FUNCTION_BLOCK FB_axis
VAR_INPUT
	//bStart							: BOOL;		
END_VAR
VAR_OUTPUT
	power	: ST_McOutputs;	
	resets	: ST_McOutputs;	
	estops	: ST_McOutputs;	
	stops	: ST_McOutputs;	
	driveResets	: ST_McOutputs;	
	diags		: ST_McOutputs;	
	diagNumber	: UDINT;
	moveRels  : ST_McOutputs;
	moveVels  : ST_McOutputs;
	moveAbses : ST_McOutputs;
	readVels	 : ST_McOutputs;
	actVel								: LREAL;
	readPoses	 : ST_McOutputs;
	actPos								: LREAL;
END_VAR
VAR_IN_OUT
	Axis: AXIS_REF;
END_VAR
VAR
	//eState		: axisState;
	mcPower		: MC_Power;
	mcReset		: MC_Reset;
	//mcDriveReset: FB_SoEReset;
	mcMoveAbs	: MC_MoveAbsolute;
	mcStop		: MC_Stop;
	mcMoveRel	: MC_MoveRelative;
	//mcReadDiag	: FB_SoEReadDiagNumber;
	mcReadVel	: MC_ReadActualVelocity;
	mcReadPos	: MC_ReadActualPosition;
	mcMoveVel	: MC_MoveVelocity;
END_VAR

(*Axis.ReadStatus();

IF axis.Status.Error THEN
	eState := ERROR;	
END_IF
	

CASE eState OF
	INIT:
	           //gHW.errAck := TRUE; 
	    mcReset.Execute := FALSE;
		mcPower.Enable := FALSE;
		mcPower.Enable_Negative:= FALSE;
		mcPower.Enable_Positive:= FALSE;
		eState := ENABLE;
		
	ENABLE:		
	         //gHW.errAck := FALSE;
		mcPower.Enable := TRUE;
		mcPower.Enable_Negative:= TRUE;
		mcPower.Enable_Positive:= TRUE;
		IF mcPower.Status THEN
			eState := READY;
		END_IF	
		
	READY:
		IF bStart THEN
			eState:= ESTOP;
		END_IF
		
	ESTOP:		
		mcMoveRel.Distance := 100;
		mcMoveRel.Velocity := 100;
		mcMoveRel.Execute := TRUE;
		IF mcMoveRel.Done THEN
			mcMoveRel.Execute := FALSE;
			eState := READY;
		END_IF	
		
	ERROR:
		mcReset.Execute := TRUE;
		         //gHW.errAck := TRUE; 
		//mcPower.Enable := FALSE;
		//mcPower.Enable_Negative:= FALSE;
		//mcPower.Enable_Positive:= FALSE;
	    IF mcReset.Done THEN
			mcReset.Execute := FALSE;	
			eState := INIT;
		//eState := DISABLED;
		END_IF
END_CASE	

mcPower(Axis:= Axis);
mcMoveRel(Axis:= Axis);
mcReset(Axis:= Axis);*)

METHOD Enable : BOOL
VAR_INPUT
	bEnable : BOOL;
END_VAR
mcPower(
	Axis := Axis,
	Enable := bEnable,
	Enable_Positive := bEnable,
	Enable_Negative := bEnable,
	BufferMode := MC_Aborting,
	Override := 100,
	Status => power.Done,
	Error => power.Error
);
END_METHOD

METHOD eStop : BOOL
VAR_INPUT
	bExecute : BOOL;
END_VAR
VAR
	EStopDeceleration		: LREAL := 5000;
	EStopJerk				: LREAL := 20000;
END_VAR
mcStop(
	Axis := Axis,
	Execute := bExecute,
	Deceleration := EStopDeceleration,
	Jerk := EStopJerk,
	Done => estops.Done
);
END_METHOD

METHOD MoveAbs : BOOL
VAR_INPUT
	bExecute 			: BOOL;
	targetAngle 		: LREAL;
	velocityIncline		: LREAL;
END_VAR
VAR	
	accelerationIncline						: LREAL := 1000;
	decelerationIncline						: LREAL := 1500;
	jerkIncline								: LREAL;
END_VAR
mcMoveAbs(	
	Axis 		:= Axis,
	Execute 	:= bExecute,	
	Position			:= targetAngle,
	Velocity 			:= velocityIncline,//cali
	Acceleration 		:= accelerationIncline,
	Deceleration 		:= decelerationIncline,
	Jerk 				:= jerkIncline,	
	Done 			=> moveAbses.Done,
	Busy 			=> moveAbses.Busy,
	Active 			=> moveAbses.Active,
	CommandAborted 	=> moveAbses.CommandAborted,
	Error 			=> moveAbses.Error,
	ErrorID 		=> moveAbses.ErrorID,	
);
END_METHOD

METHOD MoveRel : BOOL
VAR_INPUT
	bExecute : BOOL;
	relAngle : LREAL;
END_VAR
VAR
	velocityIncline							: LREAL := 100;
	accelerationIncline						: LREAL := 1000;
	decelerationIncline						: LREAL := 1500;
	jerkIncline								: LREAL;
END_VAR
mcMoveRel(
	Axis := Axis,
	Execute := bExecute,
	Distance			:= relAngle,
	Velocity 			:= velocityIncline,//cali
	Acceleration 		:= accelerationIncline,
	Deceleration 		:= decelerationIncline,
	Jerk 				:= jerkIncline,	
	Done 			=> moveRels.Done,
	Busy 			=> moveRels.Busy,
	Active 			=> moveRels.Active,
	CommandAborted 	=> moveRels.CommandAborted,
	Error 			=> moveRels.Error,
	ErrorID 		=> moveRels.ErrorID
);
END_METHOD

METHOD MoveVel : BOOL
VAR_INPUT
	bExecute 		: BOOL;
	velocity		: LREAL;
	acceleration	: LREAL;
	deceleration	: LREAL;
	jerk			: LREAL;
	Direction		: MC_Direction;
END_VAR
VAR
	//BufferMode: MC_Aborting
END_VAR
mcMoveVel(	
	Axis 		:= Axis,
	Execute 	:= bExecute,		
	Velocity 			:= velocity*1,//speedCalibrationFactorL,//cali
	Acceleration 		:= acceleration,
	Deceleration 		:= deceleration,
	Jerk 				:= jerk,	
	BufferMode 			:= MC_Aborting,
	InVelocity 		=> moveVels.Done,
	Busy 			=> moveVels.Busy,
	Active 			=> moveVels.Active,
	CommandAborted 	=> moveVels.CommandAborted,
	Error 			=> moveVels.Error,
	ErrorID 		=> moveVels.ErrorID,	
);
END_METHOD

METHOD ReadPos : BOOL
VAR_INPUT
	bEnable : BOOL;
END_VAR
mcReadPos (
	Axis := Axis,
	Enable := bEnable,
	Busy => readPoses.Busy,
	Position => ActPos
	//Error => diagNumberError,
	//AdsErrId => diagNumberAdsErrorID,
	//SercosErrId => diagNumberSercosErrorID 
);
END_METHOD

METHOD ReadVel : BOOL
VAR_INPUT
	bEnable : BOOL;
END_VAR
mcReadVel (
	Axis := Axis,
	Enable := bEnable,
	Busy => readVels.Busy,
	ActualVelocity => ActVel
	//Error => diagNumberError,
	//AdsErrId => diagNumberAdsErrorID,
	//SercosErrId => diagNumberSercosErrorID 
);
END_METHOD

METHOD Reset : BOOL
VAR_INPUT
	bExecute : BOOL;
END_VAR
mcReset(
	Axis := Axis,
	Execute := bExecute,
	Done => resets.Done,
	Error => resets.Error
);
END_METHOD

METHOD Stop : BOOL
VAR_INPUT
	bExecute : BOOL;
	Deceleration		: LREAL;
	Jerk				: LREAL;	
END_VAR
mcStop(
	Axis := Axis,
	Execute := bExecute,
	Deceleration := Deceleration,
	Jerk := Jerk,
	Done => stops.Done
);
END_METHOD

END_FUNCTION_BLOCK

(* stored: Version 1.1.0.1, ProductVersion 3.1.4024.0
   POU FB_axis: Id {4468d1f4-b80f-4453-9c9f-d05c198a1318}, SpecialFunc None
   Method Enable: Id {fafdec5a-2753-495e-9cdd-95c4346a412f}
   Method eStop: Id {02e22e27-1058-44a9-8b64-7f96890cb740}
   Method MoveAbs: Id {5bf6f79b-6023-4c7c-b620-143a2d148800}
   Method MoveRel: Id {96010620-48b2-41da-a2af-748d554297fb}
   Method MoveVel: Id {312f59aa-a034-40bb-82d8-2b12d481da77}
   Method ReadPos: Id {b789b23d-68f6-4e86-8272-36cde9f272d7}
   Method ReadVel: Id {56af1527-0690-4573-909e-0b3ac89fce64}
   Method Reset: Id {2469fb7d-06dc-40d0-95f8-bc65e9decc8a}
   Method Stop: Id {a0608013-dbe8-4f07-943e-03ad437eb627} *)
